KUKA KRL data list: SPS_CYCLE_TIME.dat

&ACCESS RV
&PARAM TEMPLATE = C:\KRC\Roboter\Template\ExpertVorgabe
&PARAM EDITMASK = *
DEFDAT sps_cycle_time PUBLIC

GLOBAL ENUM E_PROPERTY_CYCLE_TIME GET, SET
REAL rCycleTime=0.0

ENDDAT
